// Mitsubishi GX Works2 project: XY_DELTA   PLC: FX3U/FX3UC

PROGRAM MAIN
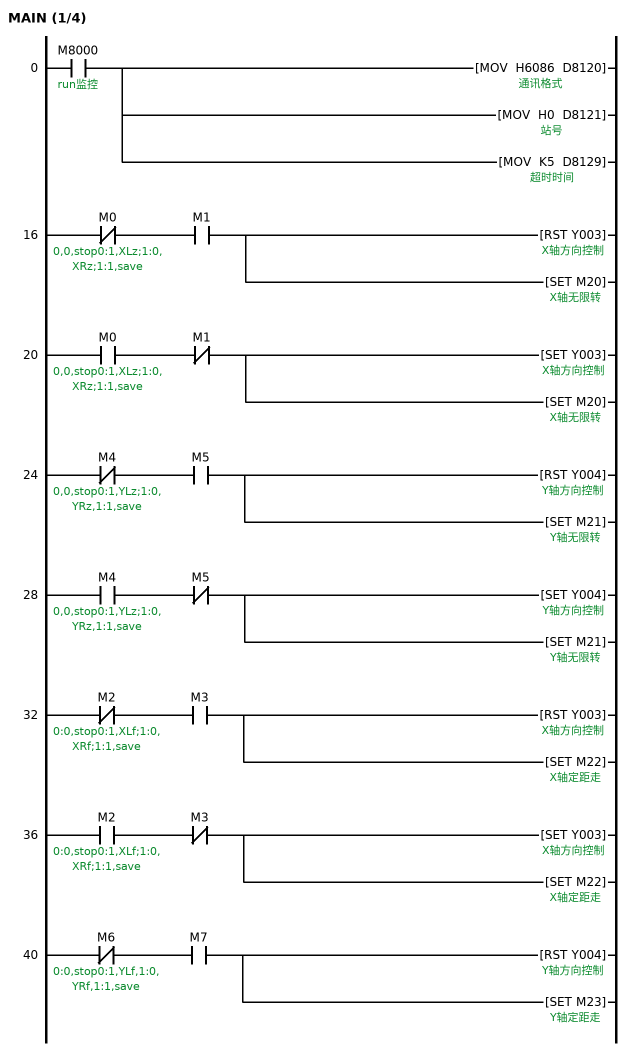
0     LD      M8000  ; run监控
      MOV     H6086 D8120  ; 通讯格式
      MOV     H0 D8121  ; 站号
      MOV     K5 D8129  ; 超时时间
16    LDI     M0  ; 0,0,stop0:1,XLz;1:0,XRz;1:1,save
      AND     M1
      RST     Y003  ; X轴方向控制
      SET     M20  ; X轴无限转
20    LD      M0  ; 0,0,stop0:1,XLz;1:0,XRz;1:1,save
      ANI     M1
      SET     Y003  ; X轴方向控制
      SET     M20  ; X轴无限转
24    LDI     M4  ; 0,0,stop0:1,YLz;1:0,YRz,1:1,save
      AND     M5
      RST     Y004  ; Y轴方向控制
      SET     M21  ; Y轴无限转
28    LD      M4  ; 0,0,stop0:1,YLz;1:0,YRz,1:1,save
      ANI     M5
      SET     Y004  ; Y轴方向控制
      SET     M21  ; Y轴无限转
32    LDI     M2  ; 0:0,stop0:1,XLf;1:0,XRf;1:1,save
      AND     M3
      RST     Y003  ; X轴方向控制
      SET     M22  ; X轴定距走
36    LD      M2  ; 0:0,stop0:1,XLf;1:0,XRf;1:1,save
      ANI     M3
      SET     Y003  ; X轴方向控制
      SET     M22  ; X轴定距走
40    LDI     M6  ; 0:0,stop0:1,YLf,1:0,YRf,1:1,save
      AND     M7
      RST     Y004  ; Y轴方向控制
      SET     M23  ; Y轴定距走
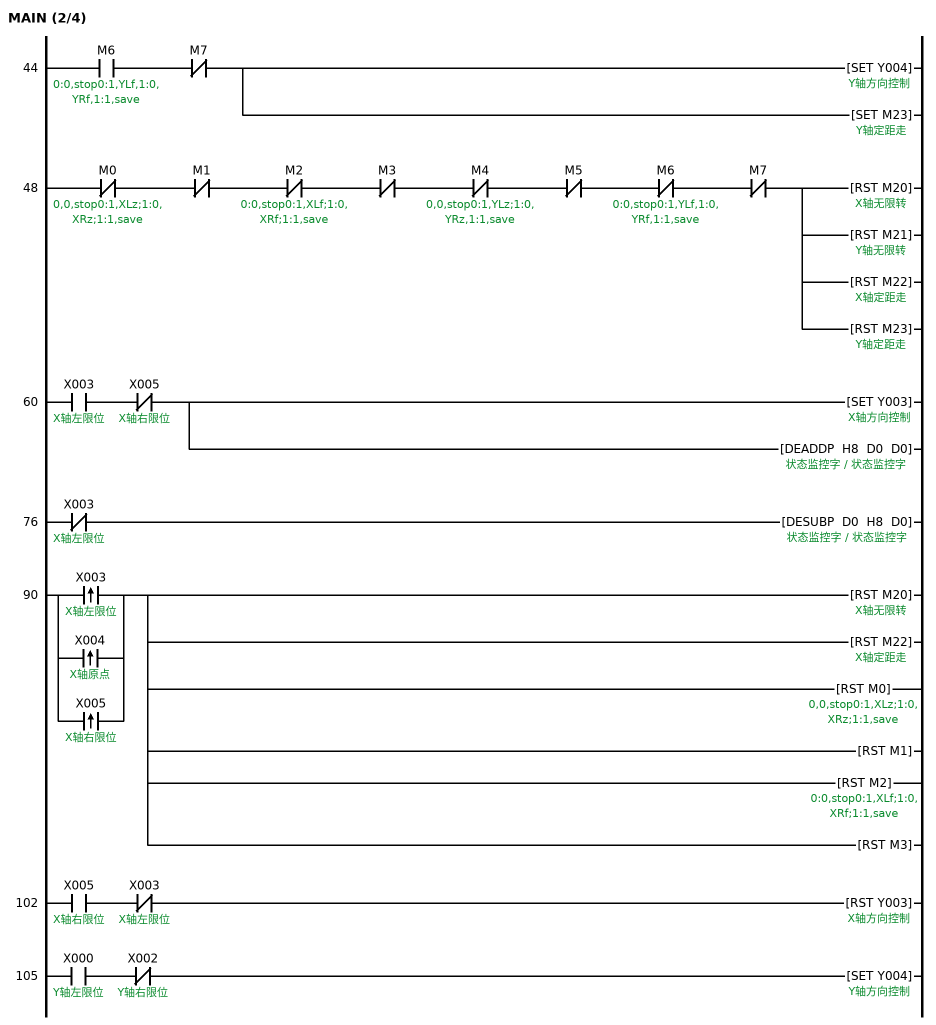
44    LD      M6  ; 0:0,stop0:1,YLf,1:0,YRf,1:1,save
      ANI     M7
      SET     Y004  ; Y轴方向控制
      SET     M23  ; Y轴定距走
48    LDI     M0  ; 0,0,stop0:1,XLz;1:0,XRz;1:1,save
      ANI     M1
      ANI     M2  ; 0:0,stop0:1,XLf;1:0,XRf;1:1,save
      ANI     M3
      ANI     M4  ; 0,0,stop0:1,YLz;1:0,YRz,1:1,save
      ANI     M5
      ANI     M6  ; 0:0,stop0:1,YLf,1:0,YRf,1:1,save
      ANI     M7
      RST     M20  ; X轴无限转
      RST     M21  ; Y轴无限转
      RST     M22  ; X轴定距走
      RST     M23  ; Y轴定距走
60    LD      X003  ; X轴左限位
      ANI     X005  ; X轴右限位
      SET     Y003  ; X轴方向控制
      DEADDP  H8 D0 D0  ; 状态监控字
76    LDI     X003  ; X轴左限位
      DESUBP  D0 H8 D0
90    LDP     X003  ; X轴左限位
      ORP     X004  ; X轴原点
      ORP     X005  ; X轴右限位
      RST     M20  ; X轴无限转
      RST     M22  ; X轴定距走
      RST     M0  ; 0,0,stop0:1,XLz;1:0,XRz;1:1,save
      RST     M1
      RST     M2  ; 0:0,stop0:1,XLf;1:0,XRf;1:1,save
      RST     M3
102   LD      X005  ; X轴右限位
      ANI     X003  ; X轴左限位
      RST     Y003  ; X轴方向控制
105   LD      X000  ; Y轴左限位
      ANI     X002  ; Y轴右限位
      SET     Y004  ; Y轴方向控制
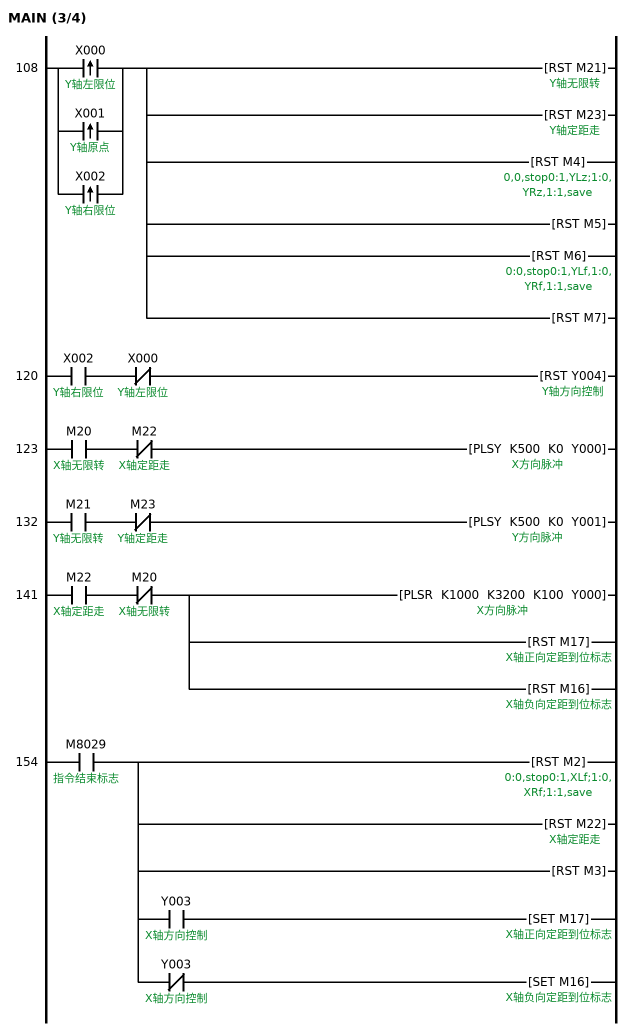
108   LDP     X000  ; Y轴左限位
      ORP     X001  ; Y轴原点
      ORP     X002  ; Y轴右限位
      RST     M21  ; Y轴无限转
      RST     M23  ; Y轴定距走
      RST     M4  ; 0,0,stop0:1,YLz;1:0,YRz,1:1,save
      RST     M5
      RST     M6  ; 0:0,stop0:1,YLf,1:0,YRf,1:1,save
      RST     M7
120   LD      X002  ; Y轴右限位
      ANI     X000  ; Y轴左限位
      RST     Y004  ; Y轴方向控制
123   LD      M20  ; X轴无限转
      ANI     M22  ; X轴定距走
      PLSY    K500 K0 Y000  ; X方向脉冲
132   LD      M21  ; Y轴无限转
      ANI     M23  ; Y轴定距走
      PLSY    K500 K0 Y001  ; Y方向脉冲
141   LD      M22  ; X轴定距走
      ANI     M20  ; X轴无限转
      PLSR    K1000 K3200 K100 Y000  ; X方向脉冲
      RST     M17  ; X轴正向定距到位标志
      RST     M16  ; X轴负向定距到位标志
154   LD      M8029  ; 指令结束标志
      RST     M2  ; 0:0,stop0:1,XLf;1:0,XRf;1:1,save
      RST     M22  ; X轴定距走
      RST     M3
      MPS
      AND     Y003  ; X轴方向控制
      SET     M17  ; X轴正向定距到位标志
      MPP
      ANI     Y003  ; X轴方向控制
      SET     M16  ; X轴负向定距到位标志
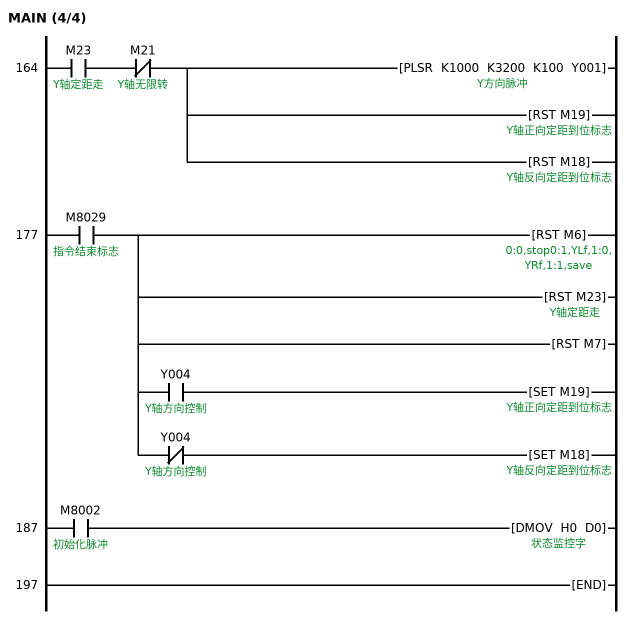
164   LD      M23  ; Y轴定距走
      ANI     M21  ; Y轴无限转
      PLSR    K1000 K3200 K100 Y001  ; Y方向脉冲
      RST     M19  ; Y轴正向定距到位标志
      RST     M18  ; Y轴反向定距到位标志
177   LD      M8029  ; 指令结束标志
      RST     M6  ; 0:0,stop0:1,YLf,1:0,YRf,1:1,save
      RST     M23  ; Y轴定距走
      RST     M7
      MPS
      AND     Y004  ; Y轴方向控制
      SET     M19  ; Y轴正向定距到位标志
      MPP
      ANI     Y004  ; Y轴方向控制
      SET     M18  ; Y轴反向定距到位标志
187   LD      M8002  ; 初始化脉冲
      DMOV    H0 D0
197   END
END_PROGRAM

// device comments not shown above
M8  ; X轴正方向
M9  ; X轴反方向
M10  ; Y轴正转
M11  ; Y轴左转
M12  ; X轴无限转
M13  ; Y轴无限转
M14  ; X轴定距走
M15  ; Y轴定距走
M24  ; X轴定距完成标志
M25  ; Y轴定距完成标志
D1  ; 中间位
